# EPICS SNL sequencer program: aptmsupervisorApp/src/dummy-old.stt
program dummy

%%#include <stdio.h>
%%#include <string.h>
%%#include <stdlib.h>

%%void printstatus(SS_ID ssId, string Msg, VAR_ID pvindex);

foreign ssId;

string myPV;
assign myPV to "testmypv:currentState";

int myPV2;
assign myPV2 to "$(P):stateOut";

ss ss1 {

    state state_one
	{
		entry
		{
			printf("We entered state one\n");
			myPV2 = 5;
			pvPut(myPV2);
		}

		when (delay(5))
		{
        } state state_two
	}

	state state_two
	{
		entry
		{
			printf("We entered state two\n");
			myPV2 = 8;
			pvPut(myPV2);

		}

		when (delay(5))
		{
		} state state_one
	}

}

%{

void printstatus(SS_ID ssId, string Msg, VAR_ID pvindex) {

	strcpy((char *)pvindex,Msg);
	seq_pvPut(ssId,pvindex,ASYNC);
	}
}%
